// TIA Portal V19 export
TYPE "LAF_typePlasticWorkstationEm5ParametersInterfaceHmi"
// stored: Access Published
   STRUCT
      configuration : "LAF_typeRollerEm1ParametersHmi";
      commands : "LBC_typeInterfaceCommands";
      monitoring { S7_SetPoint := 'True'} : "LAF_typePlasticWorkstationEm5ProcessValuesHmi";
   END_STRUCT;
END_TYPE
